FUNCTION FC_FLIP_WORD
VAR_INPUT
	In : POINTER TO BYTE;
	Out : POINTER TO BYTE;
END_VAR
VAR
	ByteArray : ARRAY[0..1] OF BYTE;
	ReturnArray : ARRAY[0..1] OF BYTE;
END_VAR

MEMCPY(srcAddr := In, destAddr := ADR(ByteArray), n := 2);

ReturnArray[0] := ByteArray[1];
ReturnArray[1] := ByteArray[0];

MEMCPY(srcAddr := ADR(ReturnArray), destAddr := Out, n := 2);

END_FUNCTION

(* stored: Version 1.1.0.1, ProductVersion 3.1.4024.12
   POU FC_FLIP_WORD: Id {7fe563d9-37f2-4556-b4ec-0bf3abbb4d07}, SpecialFunc None *)
